FUNCTION_BLOCK ServoNC IMPLEMENTS I_EncodedDrive
VAR_INPUT
	bEnable : BOOL;
END_VAR
VAR_OUTPUT	
	ready : BOOL;
	position : LREAL;
	velocity : LREAL;
END_VAR
VAR
	axis : AXIS_REF;
	
	mcReadPosition : MC_ReadActualPosition; //continuous enable FBs
	mcReadVelocity : MC_ReadActualVelocity;
	mcReadError : MC_ReadAxisError;
	mcPower : MC_Power;
	
	mcReset : MC_Reset; //rising edge FBs
	mcMoveAbsolute : MC_MoveAbsolute;
	mcMoveRelative : MC_MoveRelative;
	mcMoveVelocity : MC_MoveVelocity;
	
	mcSetPosition : MC_SetPosition;
	mcStop : MC_Stop;
END_VAR
VAR_STAT CONSTANT
	targetingVelocity : INT := 500;
	continuousVelocity : INT := 100;
END_VAR

override();

blocks();

mcReset.Execute := FALSE;
mcMoveAbsolute.Execute := FALSE;
mcMoveRelative.Execute := FALSE;
mcMoveVelocity.Execute := FALSE;
mcSetPosition.Execute := FALSE;
mcStop.Execute := FALSE;

blocks();

ready := bEnable AND NOT Active;

PROPERTY Active : BOOL
GET
Active := 
	mcMoveAbsolute.Busy OR 
	mcMoveRelative.Busy OR 
	mcMoveVelocity.Busy OR 
	mcSetPosition.Busy OR 
	mcReset.Busy OR 
	mcStop.Busy;
END_GET
END_PROPERTY

METHOD PROTECTED blocks : BOOL
mcReadPosition(
	Axis:= axis, 
	Enable:= TRUE, 
	Valid=> , 
	Busy=> , 
	Error=> , 
	ErrorID=> , 
	Position=> position);
	
mcReadVelocity(
	Axis:= axis, 
	Enable:= TRUE, 
	Valid=> , 
	Busy=> , 
	Error=> , 
	ErrorID=> , 
	ActualVelocity=> velocity);
	
mcReadError(
	Axis:= axis, 
	Enable:= TRUE, 
	Valid=> , 
	Busy=> , 
	Error=> , 
	ErrorID=> , 
	AxisErrorID=> );

mcReset(
	Axis:= axis, 
	Execute:= , 
	Done=> , 
	Busy=> , 
	Error=> , 
	ErrorID=> );

mcPower(
	Axis:= axis, 
	Enable:= bEnable, 
	Enable_Positive:= TRUE, 
	Enable_Negative:= TRUE, 
	Override:= 100, 
	BufferMode:= , 
	Options:= , 
	Status=> , 
	Busy=> , 
	Active=> , 
	Error=> , 
	ErrorID=> );

mcMoveAbsolute(
	Axis:= axis, 
	Execute:= , 
	Position:= , 
	Velocity:= targetingVelocity, 
	Acceleration:= , 
	Deceleration:= , 
	Jerk:= , 
	BufferMode:= , 
	Options:= , 
	Done=> , 
	Busy=> , 
	Active=> , 
	CommandAborted=> , 
	Error=> , 
	ErrorID=> );
	
mcMoveRelative(
	Axis:= axis, 
	Execute:= , 
	Distance:= ,
	Velocity:= targetingVelocity, 
	Acceleration:= , 
	Deceleration:= , 
	Jerk:= , 
	BufferMode:= , 
	Options:= , 
	Done=> , 
	Busy=> , 
	Active=> , 
	CommandAborted=> , 
	Error=> , 
	ErrorID=> );
	
mcMoveVelocity( //stopped with stop();
	Axis:= axis, 
	Execute:= , 
	Velocity:= continuousVelocity, 
	Acceleration:= , 
	Deceleration:= , 
	Jerk:= , 
	Direction:= , 
	BufferMode:= , 
	Options:= , 
	InVelocity=> , 
	Busy=> , 
	Active=> , 
	CommandAborted=> , 
	Error=> , 
	ErrorID=> );
	
mcSetPosition(
	Axis:= axis, 
	Execute:= , 
	Position:= , 
	Mode:= , 
	Options:= , 
	Done=> , 
	Busy=> , 
	Error=> , 
	ErrorID=> );
	
mcStop(
	Axis:= axis, 
	Execute:= , 
	Deceleration:= , 
	Jerk:= , 
	Options:= , 
	Done=> , 
	Busy=> , 
	Active=> , 
	CommandAborted=> , 
	Error=> , 
	ErrorID=> );
END_METHOD

PROPERTY CurrentPosition : LREAL
GET
CurrentPosition := position;
END_GET
SET
position := CurrentPosition;
END_SET
END_PROPERTY

PROPERTY Error : BOOL
GET
error := 
	mcMoveAbsolute.Error OR 
	mcMoveRelative.Error OR 
	mcMoveVelocity.Error OR 
	mcSetPosition.Error OR 
	mcReset.Error OR 
	mcStop.Error OR
	mcReadError.AxisErrorID > 0;
END_GET
END_PROPERTY

METHOD moveAbsolute : BOOL
VAR_INPUT
	newTarget : LREAL;
END_VAR
(*
VAR_OUTPUT
	fault : BOOL;
END_VAR
*)
IF NOT Active AND NOT error THEN
	mcMoveAbsolute.Position := newTarget;
	mcMoveAbsolute.Execute := TRUE;
END_IF

moveAbsolute := (*mcMoveAbsolute.Done AND mcMoveAbsolute.Active;*)
	position = newTarget;
END_METHOD

METHOD moveContinuous : BOOL
VAR_INPUT
	//direction : BOOL; //direction (F = inwards, T = outwards)
	newDirection : MC_Direction;
END_VAR
(*
IF mcMoveVelocity.Active THEN
	stop();
END_IF

IF NOT mcStop.Done THEN
	RETURN;
END_IF
*)
(*
IF direction THEN
	mcMoveVelocity.Direction := MC_Positive_Direction;
ELSE
	mcMoveVelocity.Direction := MC_Negative_Direction;
END_IF
*)
mcMoveVelocity.Direction := newDirection;

IF NOT mcMoveVelocity.Error THEN
	mcMoveVelocity.Execute := TRUE;
	moveContinuous := TRUE;
END_IF
END_METHOD

METHOD moveRelative : BOOL
VAR_INPUT
	distance : LREAL;
END_VAR
mcMoveRelative.Distance := distance;

moveRelative := mcMoveRelative.Done;
END_METHOD

METHOD PROTECTED override : BOOL
VAR_INPUT
END_VAR
IF error THEN
	stop();
	reset();
END_IF
END_METHOD

METHOD reset : BOOL
VAR_INPUT
END_VAR
mcReset.Execute := TRUE;

reset := mcReset.Done;
END_METHOD

METHOD setPosition : BOOL
VAR_INPUT
	newPosition : LREAL;
END_VAR
mcSetPosition.Position := newPosition;
mcSetPosition.Execute := TRUE;

setPosition := position = newPosition;
END_METHOD

METHOD stop : BOOL
VAR_INPUT
END_VAR
mcStop.Execute := TRUE;

mcMoveAbsolute.Execute := FALSE;
mcMoveRelative.Execute := FALSE;
mcMoveVelocity.Execute := FALSE;

stop := velocity = 0;
END_METHOD

PROPERTY TargetPosition : LREAL
GET
END_GET
SET
moveAbsolute(newTarget := TargetPosition);
END_SET
END_PROPERTY

END_FUNCTION_BLOCK

(* stored: Version 1.1.0.1, ProductVersion 3.1.4024.11
   POU ServoNC: Id {75aeb41f-9c42-4fdd-a248-5a35249aaeef}, SpecialFunc None
   Folder Hidden: Id {33867db6-956b-4771-8888-27808006f0f8}
   Folder Properties: Id {918a9336-51e6-4f77-b14a-277af17aec8d}
   Property Active: Id {9ca9611d-03a7-4e4a-8b86-bcafcf6f3dae}
   Get Get: Id {dc2f1cd0-2d8c-4b1a-9c1d-b817714e0852}
   Method blocks: Id {c5dfa57b-0a56-4ed3-9bb6-00ac0edd5167}
   Property CurrentPosition: Id {6c56d64e-ac1b-41ea-a0b5-4b90587e60c8}
   Get Get: Id {7f404ebf-5a45-40cc-b2c1-17d7e142d6ea}
   Set Set: Id {43ba461e-906e-4892-adc8-7161535d4c55}
   Property Error: Id {dfc53259-f873-4204-9898-7c2bcbb84bbc}
   Get Get: Id {3c92fb5b-2f0c-47d8-b261-b128d2d3839f}
   Method moveAbsolute: Id {197f1e2a-d59a-4539-a012-10c7b6cc59dc}
   Method moveContinuous: Id {dc9c1fca-c1e6-4169-9d22-4d692500a932}
   Method moveRelative: Id {23e1ffcc-9488-4a2b-aef4-34097ab1a47c}
   Method override: Id {1c62cf92-4886-4a5d-bb8d-cbbba9fb85c5}
   Method reset: Id {2d01a834-2971-4741-9f95-5e265fcf2106}
   Method setPosition: Id {f5663573-0235-4447-88d8-4f50aff4c08d}
   Method stop: Id {2554da13-cf74-479a-8ac5-10025d17adfa}
   Property TargetPosition: Id {87e3d7c2-be1c-4793-ab1b-ae5c1149660a}
   Get Get: Id {3f7f630f-c4e7-4cdf-9812-c7ac8d514f92}
   Set Set: Id {d0af1b6b-507a-41be-aa7c-ff4c644be71d} *)
